// TIA Portal project "dataLogger" (V12)

(* hardware
DEVICE "S7-1200 station_1"  SIMATIC 1200-Station
   slot 0: "S7-1200 rack"  Rack  V1.0
   slot 1: "PLC_1"  CPU 1214C DC/DC/DC  6ES7 214-1AG31-0XB0  V3.0
   slot 2: "AI4 x 13 bits_1"  6ES7 231-4HD30-0XB0  V1.0
   slot 101: "CM 1241 (RS422/485)_1"  6ES7 241-1CH31-0XB0  V1.0
*)

// ===== PLC "PLC_1"  CPU 1214C DC/DC/DC =====

VAR_GLOBAL   // PLC tag table "Default tag table"
   "Sensor_Sch4" AT %I0.0 : Bool;
   "Sensor_Sch5" AT %I0.1 : Bool;
   "Sensor_Sch7" AT %I0.2 : Bool;
   "Sensor_Jager" AT %I0.3 : Bool;
   "Sensor_Sch1" AT %I0.4 : Bool;
   "Sensor_MG320" AT %I0.5 : Bool;
   "Sensor_PG12" AT %I0.6 : Bool;
   "daytime" AT %M0.0 : Bool;
   "nighttime" AT %M0.1 : Bool;
   "Sch4_Pulse" AT %M0.2 : Bool;
   "Sch5_Pulse" AT %M0.3 : Bool;
   "Sch7_Pulse" AT %M0.4 : Bool;
   "Jager_Pulse" AT %M0.5 : Bool;
   "Sch1_Pulse" AT %M0.6 : Bool;
   "AKS" AT %M0.7 : Bool;
   "End_of_shift_Pulse" AT %M1.0 : Bool;
   "End_of_shift_Flag" AT %M1.1 : Bool;
   "Start_of_shift_Pulse" AT %M1.2 : Bool;
   "Sch4_TWs_CV" AT %MD28 : DInt;
   "Sch5_TWs_CV" AT %MD4 : DInt;
   "Sch7_TWs_CV" AT %MD8 : DInt;
   "Jager_TWs_CV" AT %MD12 : DInt;
   "Sch1_TWs_CV" AT %MD16 : DInt;
   "MG320_TWs_CV" AT %MD20 : DInt;
   "PG12_TWs_CV" AT %MD24 : DInt;
   "MG320_Pulse" AT %M1.3 : Bool;
   "PG12_Pulse" AT %M1.4 : Bool;
   "Sch4_time" AT %MD32 : DInt;
   "Sch5_time" AT %MD36 : DInt;
   "Sch7_time" AT %MD40 : DInt;
   "Jager_time" AT %MD44 : DInt;
   "Sch1_time" AT %MD48 : DInt;
   "MG320_time" AT %MD52 : DInt;
   "PG12_time" AT %MD56 : DInt;
   "System_Byte" AT %MB101 : Byte;
   "Clock_Byte" AT %MB100 : Byte;
   "Clock_1Hz" AT %M100.5 : Bool;
   "Sch4_stoptime" AT %MD60 : DInt;
   "Sch5_stoptime" AT %MD64 : DInt;
   "Sch7_stoptime" AT %MD68 : DInt;
   "Jager_stoptime" AT %MD72 : DInt;
   "Sch1_stoptime" AT %MD76 : DInt;
   "MG320_stoptime" AT %MD80 : DInt;
   "PG12_stoptime" AT %MD84 : DInt;
   "FirstScan" AT %M101.0 : Bool;
   "DiagStatusUpdate" AT %M101.1 : Bool;
   "AlwaysTRUE" AT %M101.2 : Bool;
   "AlwaysFALSE" AT %M101.3 : Bool;
   "stoptimeOffset" AT %MD102 : DInt;
   "start_Sch4" AT %M106.0 : Bool;
   "start_Sch5" AT %M106.1 : Bool;
   "start_Sch7" AT %M106.2 : Bool;
   "start_Jager" AT %M106.3 : Bool;
   "start_Sch1" AT %M106.4 : Bool;
   "start_MG320" AT %M106.5 : Bool;
   "start_PG12" AT %M106.6 : Bool;
   "Sch4_stops_CV" AT %MW108 : Int;
   "Sch5_stops_CV" AT %MW110 : Int;
   "Sch7_stops_CV" AT %MW112 : Int;
   "Jager_stops_CV" AT %MW114 : Int;
   "Sch1_stops_CV" AT %MW116 : Int;
   "MG320_stops_CV" AT %MW118 : Int;
   "PG12_stops_CV" AT %MW120 : Int;
   "MG320_hour" AT %MW122 : Int;
   "MG320_minute" AT %MW124 : Int;
   "MG320_second" AT %MW126 : Int;
   "PG12_hour" AT %MW128 : Int;
   "PG12_minute" AT %MW130 : Int;
   "PG12_second" AT %MW132 : Int;
   "Jager_hour" AT %MW134 : Int;
   "Jager_minute" AT %MW136 : Int;
   "Jager_second" AT %MW138 : Int;
   "Sch1_hour" AT %MW140 : Int;
   "Sch1_minute" AT %MW142 : Int;
   "Sch1_second" AT %MW144 : Int;
   "Sch4_hour" AT %MW146 : Int;
   "Sch4_minute" AT %MW148 : Int;
   "Sch4_second" AT %MW150 : Int;
   "Sch5_hour" AT %MW152 : Int;
   "Sch5_minute" AT %MW154 : Int;
   "Sch5_second" AT %MW156 : Int;
   "Sch7_hour" AT %MW158 : Int;
   "Sch7_minute" AT %MW160 : Int;
   "Sch7_second" AT %MW162 : Int;
END_VAR

DATA_BLOCK "Date_time_DB"   // DB1
{ S7_Optimized_Access := 'FALSE' }
VERSION : 0.1
   VAR
      date_time : DTL;
      date_time_error : DInt;
   END_VAR
BEGIN
END_DATA_BLOCK

// folder: System blocks/Program resources

DATA_BLOCK "Sch4_TWs"   // DB2
{ S7_Optimized_Access := 'FALSE' }
AUTHOR : SIMATIC
FAMILY : IEC
NAME : DCNTR
VERSION : 1.2
// stored: InstanceOfName ?
"?"
BEGIN
END_DATA_BLOCK

DATA_BLOCK "Sch5_TWs"   // DB3
{ S7_Optimized_Access := 'FALSE' }
AUTHOR : SIMATIC
FAMILY : IEC
NAME : DCNTR
VERSION : 1.2
// stored: InstanceOfName ?
"?"
BEGIN
END_DATA_BLOCK

DATA_BLOCK "Sch7_TWs"   // DB4
{ S7_Optimized_Access := 'FALSE' }
AUTHOR : SIMATIC
FAMILY : IEC
NAME : DCNTR
VERSION : 1.2
// stored: InstanceOfName ?
"?"
BEGIN
END_DATA_BLOCK

DATA_BLOCK "Jager_TWs"   // DB5
{ S7_Optimized_Access := 'FALSE' }
AUTHOR : SIMATIC
FAMILY : IEC
NAME : DCNTR
VERSION : 1.2
// stored: InstanceOfName ?
"?"
BEGIN
END_DATA_BLOCK

DATA_BLOCK "Sch1_TWs"   // DB6
{ S7_Optimized_Access := 'FALSE' }
AUTHOR : SIMATIC
FAMILY : IEC
NAME : DCNTR
VERSION : 1.2
// stored: InstanceOfName ?
"?"
BEGIN
END_DATA_BLOCK

DATA_BLOCK "Sch5_timer"   // DB7
{ S7_Optimized_Access := 'FALSE' }
AUTHOR : Simatic
FAMILY : IEC
NAME : IEC_TMR
VERSION : 1.0
// stored: InstanceOfName ?
"?"
BEGIN
END_DATA_BLOCK

DATA_BLOCK "PG12_TWs"   // DB8
{ S7_Optimized_Access := 'FALSE' }
AUTHOR : SIMATIC
FAMILY : IEC
NAME : DCNTR
VERSION : 1.2
// stored: InstanceOfName ?
"?"
BEGIN
END_DATA_BLOCK

DATA_BLOCK "IEC_Timer_0_DB"   // DB9
{ S7_Optimized_Access := 'FALSE' }
AUTHOR : Simatic
FAMILY : IEC
NAME : IEC_TMR
VERSION : 1.0
// stored: InstanceOfName ?
"?"
BEGIN
END_DATA_BLOCK

DATA_BLOCK "MG320_TWs"   // DB10
{ S7_Optimized_Access := 'FALSE' }
AUTHOR : SIMATIC
FAMILY : IEC
NAME : DCNTR
VERSION : 1.2
// stored: InstanceOfName ?
"?"
BEGIN
END_DATA_BLOCK

DATA_BLOCK "Tparo_Sch4"   // DB11
{ S7_Optimized_Access := 'FALSE' }
AUTHOR : SIMATIC
FAMILY : IEC
NAME : DCNTR
VERSION : 1.2
// stored: InstanceOfName ?
"?"
BEGIN
END_DATA_BLOCK

DATA_BLOCK "IEC_Timer_0_DB_2"   // DB12
{ S7_Optimized_Access := 'FALSE' }
AUTHOR : Simatic
FAMILY : IEC
NAME : IEC_TMR
VERSION : 1.0
// stored: InstanceOfName ?
"?"
BEGIN
END_DATA_BLOCK

DATA_BLOCK "IEC_Timer_0_DB_3"   // DB13
{ S7_Optimized_Access := 'FALSE' }
AUTHOR : Simatic
FAMILY : IEC
NAME : IEC_TMR
VERSION : 1.0
// stored: InstanceOfName ?
"?"
BEGIN
END_DATA_BLOCK

DATA_BLOCK "IEC_Timer_0_DB_4"   // DB14
{ S7_Optimized_Access := 'FALSE' }
AUTHOR : Simatic
FAMILY : IEC
NAME : IEC_TMR
VERSION : 1.0
// stored: InstanceOfName ?
"?"
BEGIN
END_DATA_BLOCK

DATA_BLOCK "IEC_Timer_0_DB_5"   // DB15
{ S7_Optimized_Access := 'FALSE' }
AUTHOR : Simatic
FAMILY : IEC
NAME : IEC_TMR
VERSION : 1.0
// stored: InstanceOfName ?
"?"
BEGIN
END_DATA_BLOCK

DATA_BLOCK "IEC_Timer_0_DB_6"   // DB16
{ S7_Optimized_Access := 'FALSE' }
AUTHOR : Simatic
FAMILY : IEC
NAME : IEC_TMR
VERSION : 1.0
// stored: InstanceOfName ?
"?"
BEGIN
END_DATA_BLOCK

DATA_BLOCK "IEC_Timer_0_DB_7"   // DB17
{ S7_Optimized_Access := 'FALSE' }
AUTHOR : Simatic
FAMILY : IEC
NAME : IEC_TMR
VERSION : 1.0
// stored: InstanceOfName ?
"?"
BEGIN
END_DATA_BLOCK

DATA_BLOCK "Sch4_timer"   // DB18
{ S7_Optimized_Access := 'FALSE' }
AUTHOR : Simatic
FAMILY : IEC
NAME : IEC_TMR
VERSION : 1.0
// stored: InstanceOfName ?
"?"
BEGIN
END_DATA_BLOCK

DATA_BLOCK "Sch7_timer"   // DB19
{ S7_Optimized_Access := 'FALSE' }
AUTHOR : Simatic
FAMILY : IEC
NAME : IEC_TMR
VERSION : 1.0
// stored: InstanceOfName ?
"?"
BEGIN
END_DATA_BLOCK

DATA_BLOCK "Jager_timer"   // DB20
{ S7_Optimized_Access := 'FALSE' }
AUTHOR : Simatic
FAMILY : IEC
NAME : IEC_TMR
VERSION : 1.0
// stored: InstanceOfName ?
"?"
BEGIN
END_DATA_BLOCK

DATA_BLOCK "Sch1_timer"   // DB21
{ S7_Optimized_Access := 'FALSE' }
AUTHOR : Simatic
FAMILY : IEC
NAME : IEC_TMR
VERSION : 1.0
// stored: InstanceOfName ?
"?"
BEGIN
END_DATA_BLOCK

DATA_BLOCK "MG320_timer"   // DB22
{ S7_Optimized_Access := 'FALSE' }
AUTHOR : Simatic
FAMILY : IEC
NAME : IEC_TMR
VERSION : 1.0
// stored: InstanceOfName ?
"?"
BEGIN
END_DATA_BLOCK

DATA_BLOCK "PG12_timer"   // DB23
{ S7_Optimized_Access := 'FALSE' }
AUTHOR : Simatic
FAMILY : IEC
NAME : IEC_TMR
VERSION : 1.0
// stored: InstanceOfName ?
"?"
BEGIN
END_DATA_BLOCK

DATA_BLOCK "Tparo_Schlatter5"   // DB24
{ S7_Optimized_Access := 'FALSE' }
AUTHOR : SIMATIC
FAMILY : IEC
NAME : DCNTR
VERSION : 1.2
// stored: InstanceOfName ?
"?"
BEGIN
END_DATA_BLOCK

DATA_BLOCK "Tparo_Sch7"   // DB25
{ S7_Optimized_Access := 'FALSE' }
AUTHOR : SIMATIC
FAMILY : IEC
NAME : DCNTR
VERSION : 1.2
// stored: InstanceOfName ?
"?"
BEGIN
END_DATA_BLOCK

DATA_BLOCK "Tparo_Jager"   // DB26
{ S7_Optimized_Access := 'FALSE' }
AUTHOR : SIMATIC
FAMILY : IEC
NAME : DCNTR
VERSION : 1.2
// stored: InstanceOfName ?
"?"
BEGIN
END_DATA_BLOCK

DATA_BLOCK "Tparo_Sch1"   // DB27
{ S7_Optimized_Access := 'FALSE' }
AUTHOR : SIMATIC
FAMILY : IEC
NAME : DCNTR
VERSION : 1.2
// stored: InstanceOfName ?
"?"
BEGIN
END_DATA_BLOCK

DATA_BLOCK "Tparo_MG320"   // DB28
{ S7_Optimized_Access := 'FALSE' }
AUTHOR : SIMATIC
FAMILY : IEC
NAME : DCNTR
VERSION : 1.2
// stored: InstanceOfName ?
"?"
BEGIN
END_DATA_BLOCK

DATA_BLOCK "Tparo_PG12"   // DB29
{ S7_Optimized_Access := 'FALSE' }
AUTHOR : SIMATIC
FAMILY : IEC
NAME : DCNTR
VERSION : 1.2
// stored: InstanceOfName ?
"?"
BEGIN
END_DATA_BLOCK

DATA_BLOCK "Sch4_stops"   // DB30
{ S7_Optimized_Access := 'FALSE' }
AUTHOR : Simatic
FAMILY : IEC
NAME : CNTR
VERSION : 1.0
// stored: InstanceOfName ?
"?"
BEGIN
END_DATA_BLOCK

DATA_BLOCK "Sch5_stops"   // DB31
{ S7_Optimized_Access := 'FALSE' }
AUTHOR : Simatic
FAMILY : IEC
NAME : CNTR
VERSION : 1.0
// stored: InstanceOfName ?
"?"
BEGIN
END_DATA_BLOCK

DATA_BLOCK "Sch7_stops"   // DB32
{ S7_Optimized_Access := 'FALSE' }
AUTHOR : Simatic
FAMILY : IEC
NAME : CNTR
VERSION : 1.0
// stored: InstanceOfName ?
"?"
BEGIN
END_DATA_BLOCK

DATA_BLOCK "Jager_stops"   // DB33
{ S7_Optimized_Access := 'FALSE' }
AUTHOR : Simatic
FAMILY : IEC
NAME : CNTR
VERSION : 1.0
// stored: InstanceOfName ?
"?"
BEGIN
END_DATA_BLOCK

DATA_BLOCK "Sch1_stops"   // DB34
{ S7_Optimized_Access := 'FALSE' }
AUTHOR : Simatic
FAMILY : IEC
NAME : CNTR
VERSION : 1.0
// stored: InstanceOfName ?
"?"
BEGIN
END_DATA_BLOCK

DATA_BLOCK "MG320"   // DB35
{ S7_Optimized_Access := 'FALSE' }
AUTHOR : Simatic
FAMILY : IEC
NAME : CNTR
VERSION : 1.0
// stored: InstanceOfName ?
"?"
BEGIN
END_DATA_BLOCK

DATA_BLOCK "PG12_stops"   // DB36
{ S7_Optimized_Access := 'FALSE' }
AUTHOR : Simatic
FAMILY : IEC
NAME : CNTR
VERSION : 1.0
// stored: InstanceOfName ?
"?"
BEGIN
END_DATA_BLOCK

// folder: (top level)

FUNCTION "Activity_register" : Void   // FC1, LAD
TITLE = Counters for all welding machine
{ S7_Optimized_Access := 'FALSE' }
VERSION : 0.1
// At the end of shift, counters reset by python's AKS.
BEGIN
END_FUNCTION

FUNCTION "Reset_start_times" : Void   // FC2, LAD
{ S7_Optimized_Access := 'FALSE' }
VERSION : 0.1
BEGIN

REGION Network 1: MG320
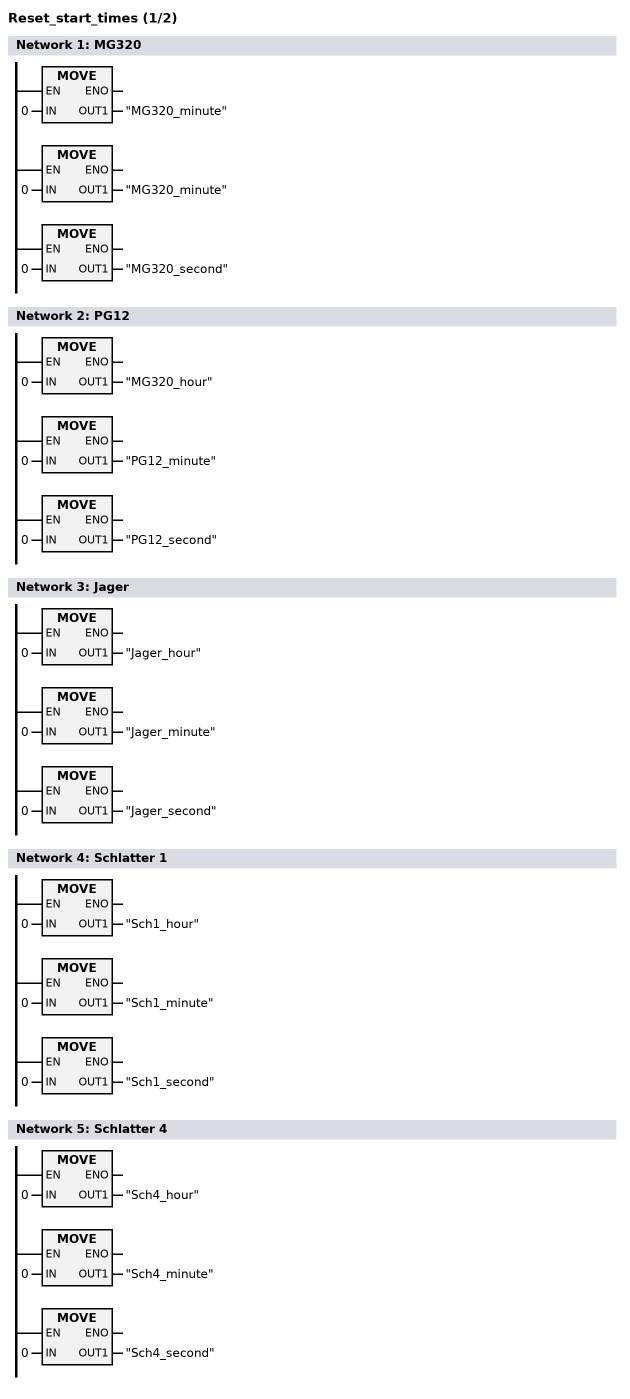
   RUNG wire#powerrail
      { S7_GenerateENO := "TRUE" } Move(in := 0, out1 => "MG320_minute")
   END_RUNG
   RUNG wire#powerrail
      { S7_GenerateENO := "TRUE" } Move(in := 0, out1 => "MG320_minute")
   END_RUNG
   RUNG wire#powerrail
      { S7_GenerateENO := "TRUE" } Move(in := 0, out1 => "MG320_second")
   END_RUNG
   // the same network as SCL:
   "MG320_minute" := 0;
   "MG320_minute" := 0;
   "MG320_second" := 0;
END_REGION

REGION Network 2: PG12
   RUNG wire#powerrail
      { S7_GenerateENO := "TRUE" } Move(in := 0, out1 => "MG320_hour")
   END_RUNG
   RUNG wire#powerrail
      { S7_GenerateENO := "TRUE" } Move(in := 0, out1 => "PG12_minute")
   END_RUNG
   RUNG wire#powerrail
      { S7_GenerateENO := "TRUE" } Move(in := 0, out1 => "PG12_second")
   END_RUNG
   // the same network as SCL:
   "MG320_hour" := 0;
   "PG12_minute" := 0;
   "PG12_second" := 0;
END_REGION

REGION Network 3: Jager
   RUNG wire#powerrail
      { S7_GenerateENO := "TRUE" } Move(in := 0, out1 => "Jager_hour")
   END_RUNG
   RUNG wire#powerrail
      { S7_GenerateENO := "TRUE" } Move(in := 0, out1 => "Jager_minute")
   END_RUNG
   RUNG wire#powerrail
      { S7_GenerateENO := "TRUE" } Move(in := 0, out1 => "Jager_second")
   END_RUNG
   // the same network as SCL:
   "Jager_hour" := 0;
   "Jager_minute" := 0;
   "Jager_second" := 0;
END_REGION

REGION Network 4: Schlatter 1
   RUNG wire#powerrail
      { S7_GenerateENO := "TRUE" } Move(in := 0, out1 => "Sch1_hour")
   END_RUNG
   RUNG wire#powerrail
      { S7_GenerateENO := "TRUE" } Move(in := 0, out1 => "Sch1_minute")
   END_RUNG
   RUNG wire#powerrail
      { S7_GenerateENO := "TRUE" } Move(in := 0, out1 => "Sch1_second")
   END_RUNG
   // the same network as SCL:
   "Sch1_hour" := 0;
   "Sch1_minute" := 0;
   "Sch1_second" := 0;
END_REGION

REGION Network 5: Schlatter 4
   RUNG wire#powerrail
      { S7_GenerateENO := "TRUE" } Move(in := 0, out1 => "Sch4_hour")
   END_RUNG
   RUNG wire#powerrail
      { S7_GenerateENO := "TRUE" } Move(in := 0, out1 => "Sch4_minute")
   END_RUNG
   RUNG wire#powerrail
      { S7_GenerateENO := "TRUE" } Move(in := 0, out1 => "Sch4_second")
   END_RUNG
   // the same network as SCL:
   "Sch4_hour" := 0;
   "Sch4_minute" := 0;
   "Sch4_second" := 0;
END_REGION

REGION Network 6: Schlatter 5
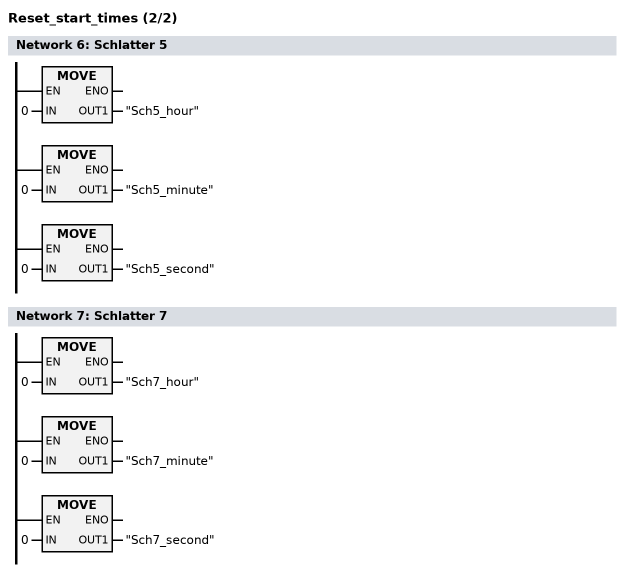
   RUNG wire#powerrail
      { S7_GenerateENO := "TRUE" } Move(in := 0, out1 => "Sch5_hour")
   END_RUNG
   RUNG wire#powerrail
      { S7_GenerateENO := "TRUE" } Move(in := 0, out1 => "Sch5_minute")
   END_RUNG
   RUNG wire#powerrail
      { S7_GenerateENO := "TRUE" } Move(in := 0, out1 => "Sch5_second")
   END_RUNG
   // the same network as SCL:
   "Sch5_hour" := 0;
   "Sch5_minute" := 0;
   "Sch5_second" := 0;
END_REGION

REGION Network 7: Schlatter 7
   RUNG wire#powerrail
      { S7_GenerateENO := "TRUE" } Move(in := 0, out1 => "Sch7_hour")
   END_RUNG
   RUNG wire#powerrail
      { S7_GenerateENO := "TRUE" } Move(in := 0, out1 => "Sch7_minute")
   END_RUNG
   RUNG wire#powerrail
      { S7_GenerateENO := "TRUE" } Move(in := 0, out1 => "Sch7_second")
   END_RUNG
   // the same network as SCL:
   "Sch7_hour" := 0;
   "Sch7_minute" := 0;
   "Sch7_second" := 0;
END_REGION
END_FUNCTION

ORGANIZATION_BLOCK "Main"   // OB1, LAD, ProgramCycle
TITLE = "Main Program Sweep (Cycle)"
{ S7_Optimized_Access := 'FALSE' }
VERSION : 0.1
BEGIN
END_ORGANIZATION_BLOCK